// SIMATIC S7-200 project (STEP 7-Micro/WIN), CPU 224 CN REL 02.01

ORGANIZATION_BLOCK MAIN:OB1
TITLE=程序注释：浙江天煌科技实业有限公司       http://www.tianhuang.cn          
// 文件名：led数码显示                                            
// 创建人：黄庆国                                                      
// 创建日期：2005.9.21                                                   
// 修改日期：                 
//                                                                                                                                                                                   版本号：V1.0
BEGIN
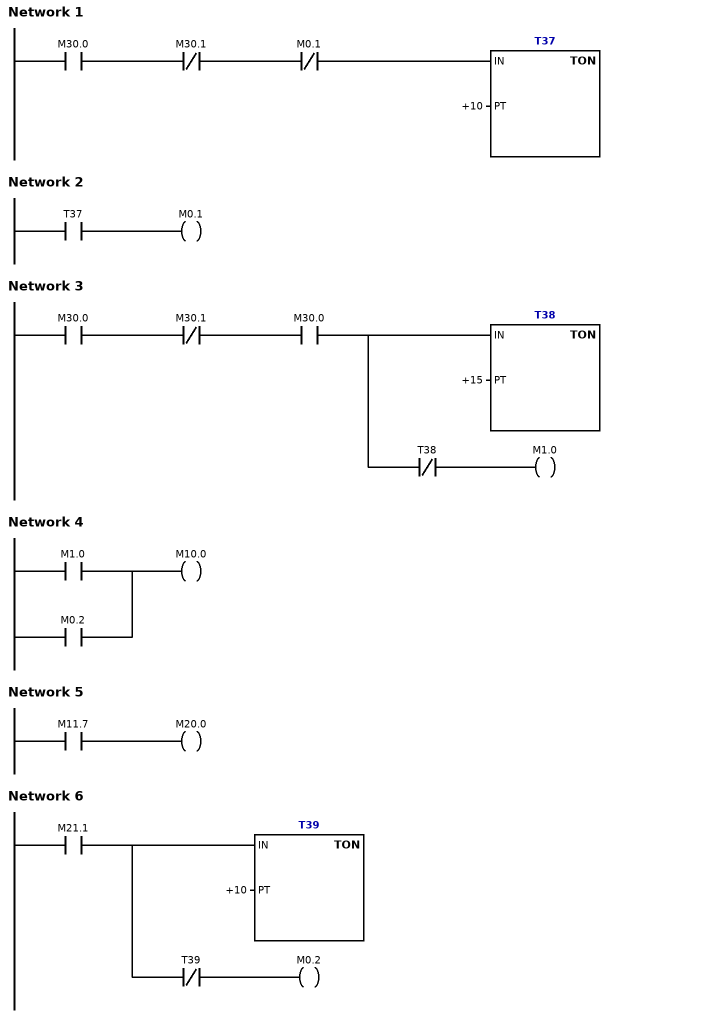
Network 1
LD     M30.0
AN     M30.1
AN     M0.1
TON    T37, +10
Network 2
LD     T37
=      M0.1
Network 3
LD     M30.0
AN     M30.1
A      M30.0
TON    T38, +15
AN     T38
=      M1.0
Network 4
LD     M1.0
O      M0.2
=      M10.0
Network 5
LD     M11.7
=      M20.0
Network 6
LD     M21.1
TON    T39, +10
AN     T39
=      M0.2
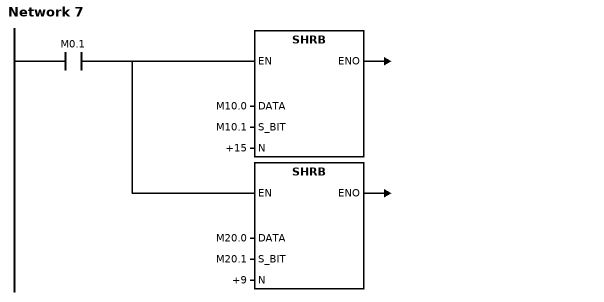
Network 7
LD     M0.1
SHRB   M10.0, M10.1, +15
SHRB   M20.0, M20.1, +9
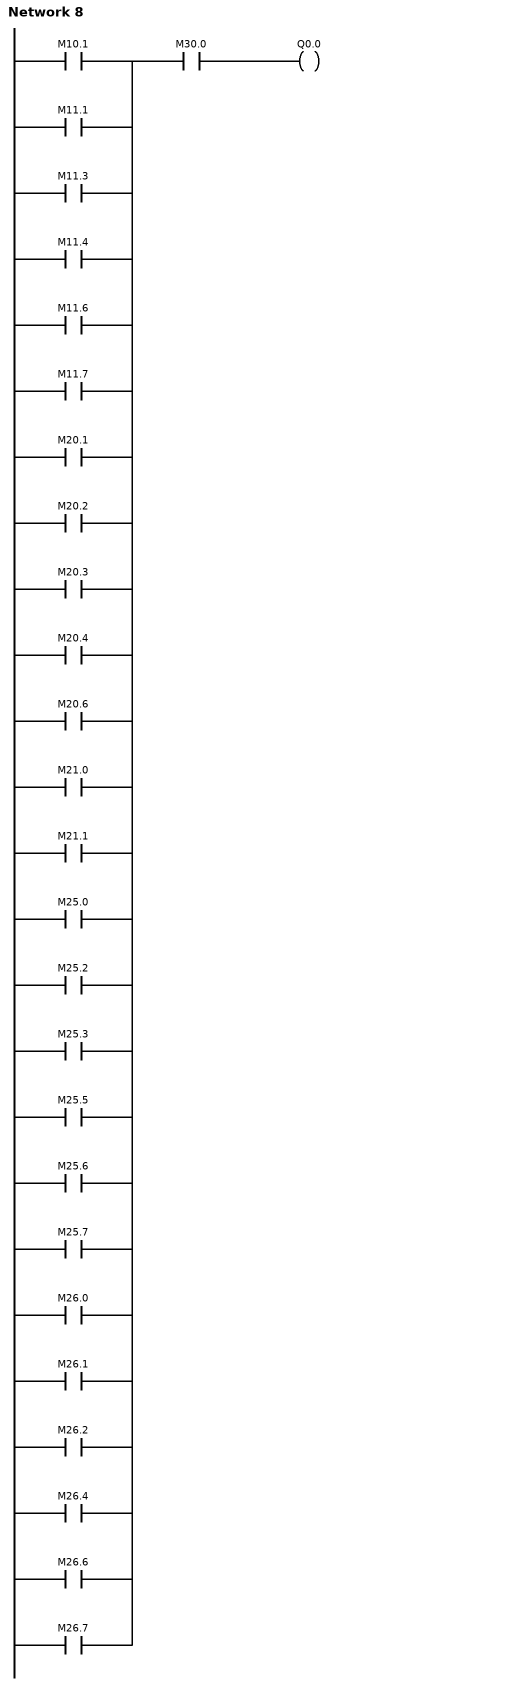
Network 8
LD     M10.1
O      M11.1
O      M11.3
O      M11.4
O      M11.6
O      M11.7
O      M20.1
O      M20.2
O      M20.3
O      M20.4
O      M20.6
O      M21.0
O      M21.1
O      M25.0
O      M25.2
O      M25.3
O      M25.5
O      M25.6
O      M25.7
O      M26.0
O      M26.1
O      M26.2
O      M26.4
O      M26.6
O      M26.7
A      M30.0
=      Q0.0
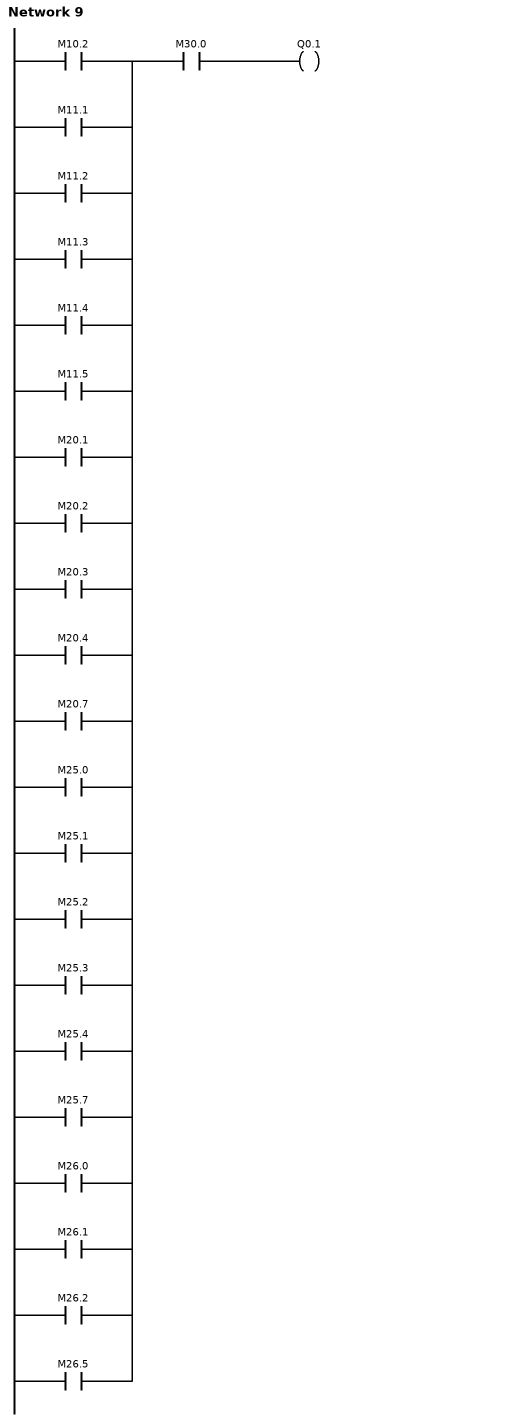
Network 9
LD     M10.2
O      M11.1
O      M11.2
O      M11.3
O      M11.4
O      M11.5
O      M20.1
O      M20.2
O      M20.3
O      M20.4
O      M20.7
O      M25.0
O      M25.1
O      M25.2
O      M25.3
O      M25.4
O      M25.7
O      M26.0
O      M26.1
O      M26.2
O      M26.5
A      M30.0
=      Q0.1
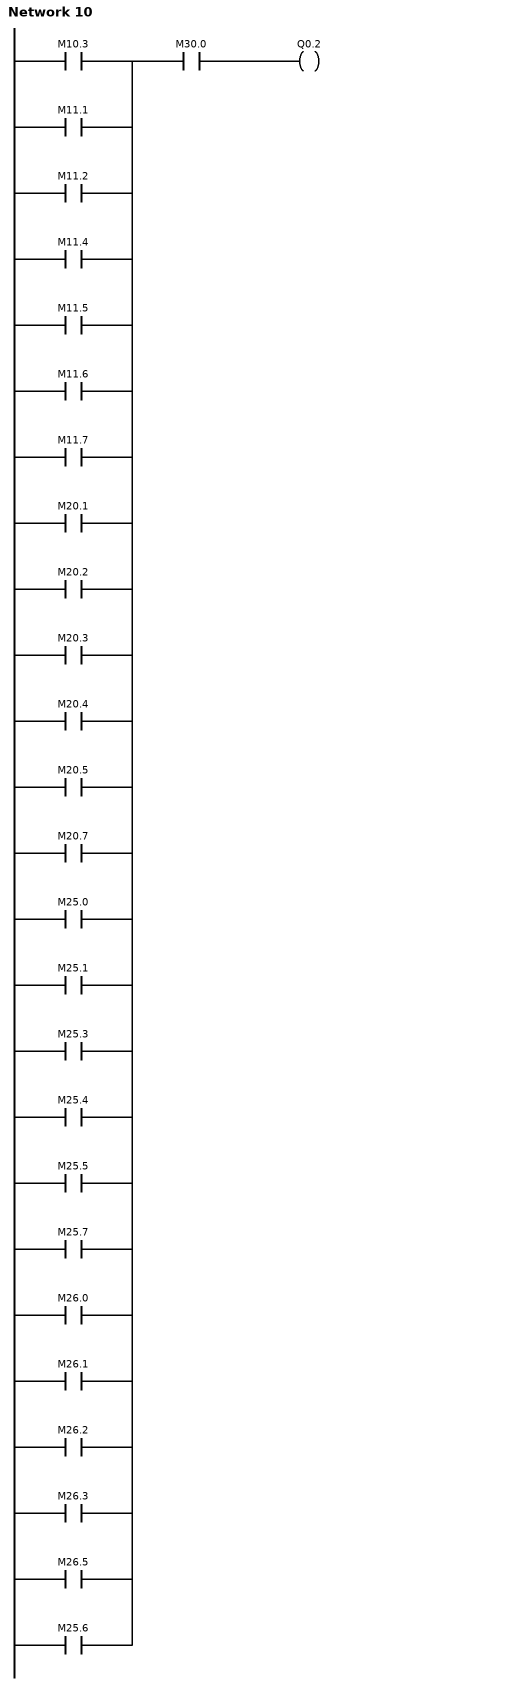
Network 10
LD     M10.3
O      M11.1
O      M11.2
O      M11.4
O      M11.5
O      M11.6
O      M11.7
O      M20.1
O      M20.2
O      M20.3
O      M20.4
O      M20.5
O      M20.7
O      M25.0
O      M25.1
O      M25.3
O      M25.4
O      M25.5
O      M25.7
O      M26.0
O      M26.1
O      M26.2
O      M26.3
O      M26.5
O      M25.6
A      M30.0
=      Q0.2
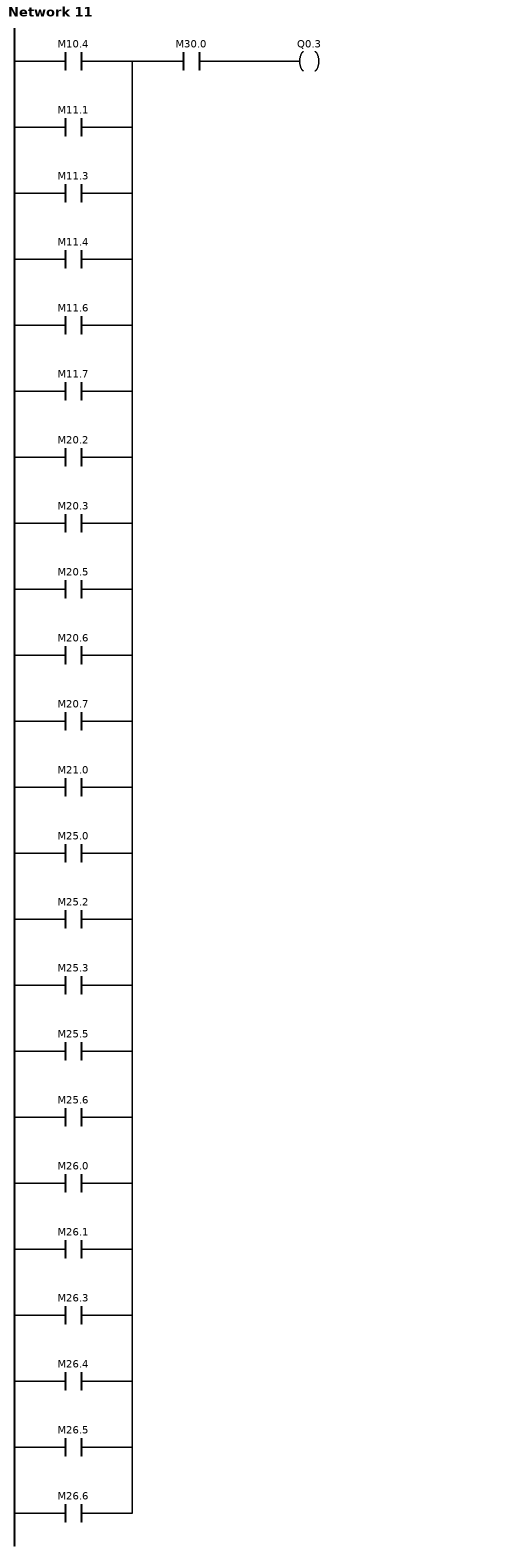
Network 11
LD     M10.4
O      M11.1
O      M11.3
O      M11.4
O      M11.6
O      M11.7
O      M20.2
O      M20.3
O      M20.5
O      M20.6
O      M20.7
O      M21.0
O      M25.0
O      M25.2
O      M25.3
O      M25.5
O      M25.6
O      M26.0
O      M26.1
O      M26.3
O      M26.4
O      M26.5
O      M26.6
A      M30.0
=      Q0.3
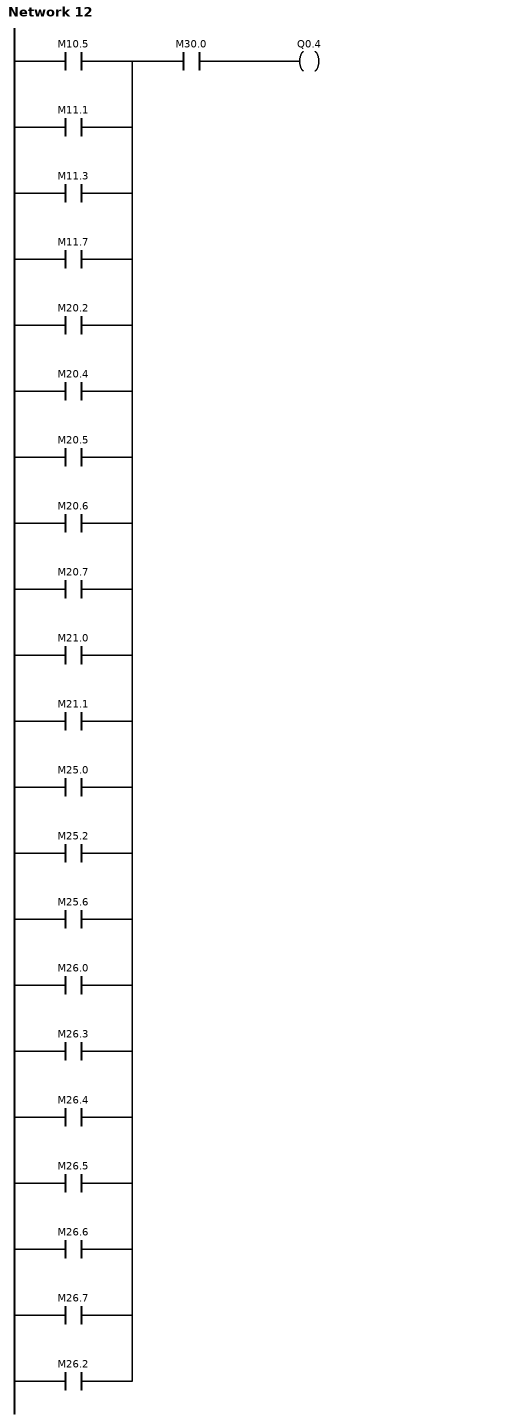
Network 12
LD     M10.5
O      M11.1
O      M11.3
O      M11.7
O      M20.2
O      M20.4
O      M20.5
O      M20.6
O      M20.7
O      M21.0
O      M21.1
O      M25.0
O      M25.2
O      M25.6
O      M26.0
O      M26.3
O      M26.4
O      M26.5
O      M26.6
O      M26.7
O      M26.2
A      M30.0
=      Q0.4
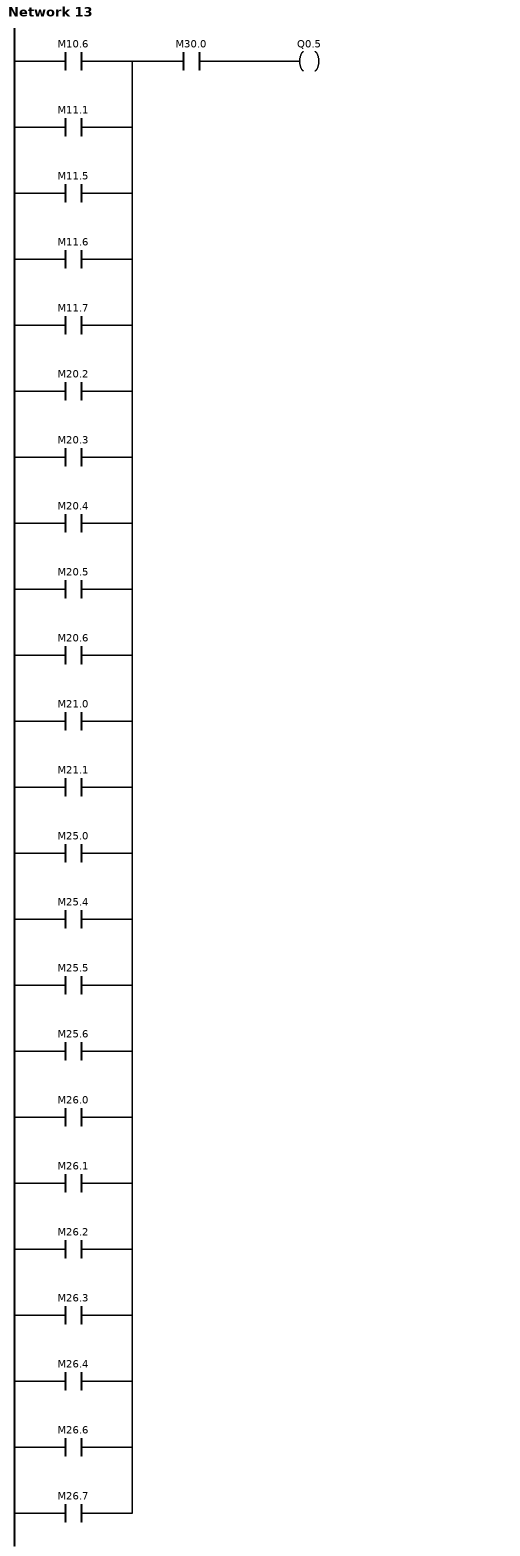
Network 13
LD     M10.6
O      M11.1
O      M11.5
O      M11.6
O      M11.7
O      M20.2
O      M20.3
O      M20.4
O      M20.5
O      M20.6
O      M21.0
O      M21.1
O      M25.0
O      M25.4
O      M25.5
O      M25.6
O      M26.0
O      M26.1
O      M26.2
O      M26.3
O      M26.4
O      M26.6
O      M26.7
A      M30.0
=      Q0.5
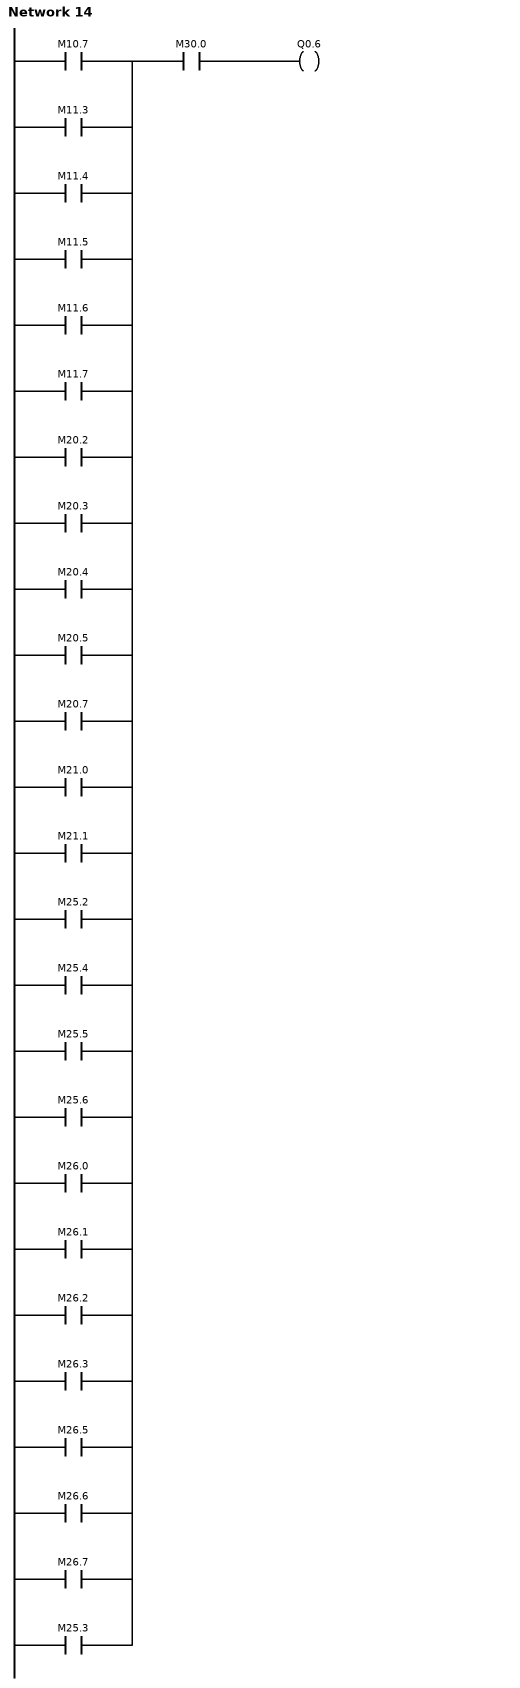
Network 14
LD     M10.7
O      M11.3
O      M11.4
O      M11.5
O      M11.6
O      M11.7
O      M20.2
O      M20.3
O      M20.4
O      M20.5
O      M20.7
O      M21.0
O      M21.1
O      M25.2
O      M25.4
O      M25.5
O      M25.6
O      M26.0
O      M26.1
O      M26.2
O      M26.3
O      M26.5
O      M26.6
O      M26.7
O      M25.3
A      M30.0
=      Q0.6
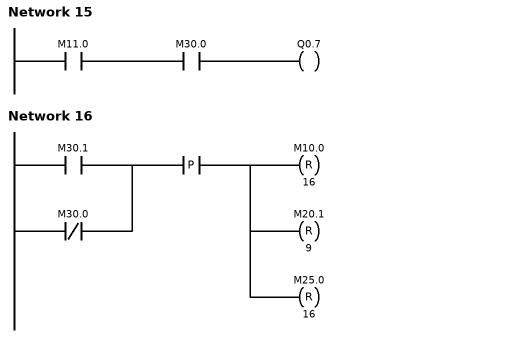
Network 15
LD     M11.0
A      M30.0
=      Q0.7
Network 16
LD     M30.1
ON     M30.0
EU
R      M10.0, 16
R      M20.1, 9
R      M25.0, 16
END_ORGANIZATION_BLOCK
